# EPICS autosave request: iocBoot/ioc13idd_LVP/auto_positions.req
file "Galil_positions.req",   P=$(P)
